(************************************************************************************)
(*							Beckhoff Automation Poland								*)
(*							F_8BYTES_TO_LREAL v1.0									*)
(*									3.07.2015										*)
(*					Funkcja zamieniająca 8 zmiennych typu BYTE na LREAL 			*)
(*__________________________________________________________________________________*)
FUNCTION F_8BYTES_TO_LREAL : LREAL
VAR_INPUT
	BByte0		: BYTE;
	BByte1		: BYTE;
	BByte2		: BYTE;
	BByte3		: BYTE;
	BByte4		: BYTE;
	BByte5		: BYTE;
	BByte6		: BYTE;
	BByte7		: BYTE;
END_VAR
VAR
	arrByte	: ARRAY [1..8] OF BYTE;
END_VAR

arrByte[1] := BByte0;
arrByte[2] := BByte1;
arrByte[3] := BByte2;
arrByte[4] := BByte3;
arrByte[5] := BByte4;
arrByte[6] := BByte5;
arrByte[7] := BByte6;
arrByte[8] := BByte7;

MEMCPY(ADR(F_8BYTES_TO_LREAL),ADR(arrByte), 8);

END_FUNCTION

(* stored: Version 1.1.0.1, ProductVersion 3.1.4026.13, FileIdentifier da5da4c4c6bdf5c65192c29a07eeade502b26abd, FileSignature 14af68694811517f181c70fb2d89fed33dbadeab46aaf40cb03c3ff66139feb37c392a9a47cdc610093f44ba3143a2c755400ef2b91092c697e42c936fa2bf9addfe3dfe5ab6dc9af5623e2671e22225b687e692079c1a32a0faf5d18978127c02aaaad09f02080da0a0d60abbbae677358350af866d7735ac869ce3c04b85b700689b2364f2aebd35238de67866fbffdf437a57656db270c90aa39ab60ca96659b469e4bbdb29916b645c6910053a7ccf956f93986c422fd14b5deba29884c7d0306a3622c613ccdbd49054c3016ebbc7f0a7a6bae2e71e316e64f0c2c68cc4b1e8efed9ed4d380a8a6cce5c37650057a909cd59e09dae10618f056540e1a16
   POU F_8BYTES_TO_LREAL: Id {54cbca58-a432-4037-a091-dfebc543201a}, SpecialFunc None *)
